{region '#Template'}
	{attribute 'Version' := '5.0.0.0'}
	{attribute 'Tags' := '"LCID": "1031", "Text": "DUT, Types, Publisher, Subscriber, Global, General, Alarms, Events"'}
	{attribute 'Tags' := '"LCID": "1033", "Text": "DUT, Types, Publisher, Subscriber, Global, General, Alarms, Events"'}
	{attribute 'Description' := '"LCID": "1031", "Text": "Globale Alarme und Events"'}
	{attribute 'Description' := '"LCID": "1033", "Text": "Global alarms and events"'}
{endregion}
TYPE ST_BA_GlobalAlarmsEvents :
STRUCT
	bBurglary				: BOOL;
	bFireAlert				: BOOL;
	bCentralOff				: BOOL;
	bForcedVentilation		: BOOL;
	bAlarm1					: BOOL;
	bAlarm2					: BOOL;
	bAlarm3					: BOOL;
	bEvent1					: BOOL;
	bEvent2					: BOOL;
	bEvent3					: BOOL;
   {attribute 'hide'}
	aDummy					: ARRAY[1..6] OF BYTE; 		// padding bytes, in order to reach a limit corresponding to the largest data type (divisible by 8 bytes)
END_STRUCT
END_TYPE

(* stored: Version 1.1.0.1, ProductVersion 3.1.4024.12
   DUT ST_BA_GlobalAlarmsEvents: Id {2eea1ac1-dbeb-4010-aacd-39da6b2f2823} *)
